{attribute 'GeneratedUsingTerminal: EK1100-0000-0018'}
{attribute addProperty BoxType "EK1100-0000-0018"}
{attribute addProperty Id "Beckhoff_EQ3xxxEK1122Beckhoff_EQ3xxxEK1122_A07497C8606"}
{attribute addProperty CRC "874096031"}
{attribute addProperty Size "606"}
TYPE Beckhoff_EQ3xxx_3419A59F EXTENDS EK1100_1FC0878B :
STRUCT
	{attribute addProperty Name "Beckhoff_EQ3xxxEK1122"}
	{attribute addProperty PreviousPort "Beckhoff EQ3xxx : B"}
	Beckhoff_EQ3xxxEK1122 : Beckhoff_EQ3xxxEK1122_A07497C8;
END_STRUCT
END_TYPE

(* stored: Version 1.2.0.0, ProductVersion 3.1.4024.9
   DUT Beckhoff_EQ3xxx_3419A59F: Id {f4486b5d-ac53-4d0b-9192-6876629d3ee7} *)
